(* PLC project Generated.project, CODESYS CODESYS V3.5 SP19 Patch 1 *)
(* stored: creationDateTime 2026-09-06T13:00:42.357406, modificationDateTime 2026-09-06T13:00:42.357406 *)

(* ======================================================================= 🔌 ST_ContactorCheck — Double vérification commande/retour contacteur ─────────────────────────────────────────────────────────────── 🎯 Rôle : Structure de diagnostic pour vérification commande vs retour 📊 Diagnostic : Détection des défauts contacteur (StuckClosed / StuckOpen) 📄 Doc métier : DOC/AF/AF_Partie-03_Contrats_Composants_v2.3.md §2 ======================================================================= *)
TYPE ST_ContactorCheck : STRUCT
  Command : BOOL;  (* Ordre envoyé au contacteur (TRUE = fermé/actif) *)
  Feedback : BOOL;  (* Retour d'état câblé (TRUE = effectivement fermé) *)
  StuckClosed : BOOL;  (* Diag : commande OFF mais retour ON depuis trop longtemps → PowerCutOff *)
  StuckOpen : BOOL;  (* Diag : commande ON mais retour OFF depuis trop longtemps *)
END_STRUCT;
END_TYPE

(* ======================================================================= 🧩 ST_Fault — Brique socle défaut (2 vues : live + latchée) ─────────────────────────────────────────────────────────────── 🎯 Rôle : porter l'état défaut d'un composant, applicable dans TOUS les cas (acquittable ou non), sans brique warning séparée. • Vue LIVE (Error / ErrorId) : suit la cause, retombe seule à 0. • Vue LATCHÉE (Latched / LatchedId): mémorisée au défaut, reste jusqu'au front Reset. Le choix acquittable / non-acquittable se fait PAR CAUSE (ST_FaultCause.Latching), jamais par bloc. 🔒 Sécurité : interlock TOUJOURS sur la cause brute (Error / ErrorId), jamais sur l'acquittement. Reset TOUJOURS effectif, jamais conditionné (std §9). 🧬 Composition : brique de base réutilisable — sortie de FB, struct métier, GVL. Texte IHM NON stocké ici : dérivé côté IHM depuis LatchedId / ErrorId. 📄 Doc : DOC/STDS/CODE_QUALITY_STANDARDS.md §2quinquies / §9 ======================================================================= *)
TYPE ST_Fault : STRUCT
  Error : BOOL;  (* <-- [DIAG] vue LIVE : au moins une cause présente maintenant *)
  ErrorId : WORD;  (* <-- [DIAG] bitfield des causes présentes maintenant (0 si aucune) *)
  Latched : BOOL;  (* <-- [DIAG] vue LATCHÉE : défaut non acquitté, reste jusqu'au front Reset *)
  LatchedId : WORD;  (* <-- [DIAG] ErrorId figé à l'apparition du défaut, effacé au Reset *)
END_STRUCT;
END_TYPE

(* ======================================================================= 🧩 ST_FaultCause — Cause élémentaire alimentant ST_Fault (socle FB_FaultCore) ─────────────────────────────────────────────────────────────── 🎯 Rôle : une cause exprimée EN CLAIR (BOOL + libellé), sans bitfield ni masque. Le FB métier remplit une liste (ARRAY[0..15] OF ST_FaultCause) ; le socle FB_FaultCore en déduit ST_Fault (vue live + vue latchée). 🔒 Sécurité : interlock TOUJOURS sur Active (cause brute), jamais sur le latch. Latching = TRUE → la cause ARME la vue latchée (défaut à acquitter). Latching = FALSE → la cause n'alimente que la vue live (retombe seule). Fail-safe : une cause laissée à Latching=FALSE reste visible en live — pour la rendre acquittable, il faut le déclarer explicitement. 📄 Doc : DOC/STDS/CODE_QUALITY_STANDARDS.md §2quinquies / §9 ======================================================================= *)
TYPE ST_FaultCause : STRUCT
  Active : BOOL;  (* 1 = cause présente maintenant (interlock sur cette valeur) *)
  Latching : BOOL;  (* 1 = cause à acquitter (arme Latched) ; 0 = live seulement *)
  Texte : STRING;  (* libellé prêt IHM (non stocké dans ST_Fault, dérivé côté IHM) *)
END_STRUCT;
END_TYPE

(* ======================================================================= 🛡️ FB_Brake — Séquence frein à manque de courant (temps physiques) ─────────────────────────────────────────────────────────────── 🎯 Rôle : Gestion temporisée ouverture/fermeture frein à manque de courant 🔒 Polarité : Sécurité positive (BrakeCmd=FALSE = frein collé au repos) 🔌 Interface : Double vérification retour contacteur (ST_ContactorCheck) 📄 Doc métier : DOC/AF/AF_Partie-10_Fonction_Winch_v2.1.md §3 ======================================================================= *)
FUNCTION_BLOCK FB_Brake
  VAR_INPUT
    Enable : BOOL;  (* === COMMANDES ET CONSIGNES === --> [CMD] Autorisation generale (FALSE = frein colle) *)
    Reset : BOOL;  (* --> [CMD] Acquittement defaut (front) *)
    MovementRequested : BOOL;  (* --> [CMD] Demande de mouvement (sens+palier actifs) *)
    ContactorFeedback : BOOL;  (* === RETOURS MATERIELS & SIMULATION === --> [HW] Retour contacteur frein (TRUE = relache/ouvert) *)
    BypassContactorCheck : BOOL;  (* --> [TST] Bypass controle contacteur (simu) *)
    DelayContactClose : TIME := TIME#100ms;  (* === TEMPORISATIONS ET REGLAGES === --> [CFG] Temps de fermeture contacteur de puissance *)
    DelayMagnetise : TIME := TIME#300ms;  (* --> [CFG] Delai magnetisation moteur avant ouverture frein *)
    DelayMotorDecel : TIME := TIME#500ms;  (* --> [CFG] Delai deceleration avant collage frein *)
    FeedbackTimeout : TIME := TIME#1s0ms;  (* --> [CFG] Delai max coherence commande/retour frein *)
  END_VAR
  VAR_OUTPUT
    Ready : BOOL;  (* === ETATS IEC & DERIVATION === <-- [STAT] FB pret a fonctionner *)
    Fault : ST_Fault;  (* 🧩 Statut transverse (forme cible ST_Fault) *)
    BrakeCmd : BOOL;  (* === COMMANDES ET CONFIRMATIONS === <-- [ACT] Commande bobine frein (TRUE = relache/ouvert) *)
    BrakeCommandOpenConfirmed : BOOL;  (* <-- [STAT] Confirmation ouverture frein pour verrous *)
    ContactorCheck : ST_ContactorCheck;  (* <-- [DIAG] Diagnostic detaille retour contacteur *)
  END_VAR
  VAR
    ResetEdge : R_TRIG;  (* === TRIGGERS ET DETECTION FRONTS === . [LOC] Detecteur front acquittement *)
    BypassEdge : R_TRIG;  (* . [LOC] Detecteur front activation bypass *)
    TonMagnetise : TON;  (* === TEMPORISATEURS INTERNES === . [LOC] Temporisation avant relachement frein *)
    TonDecel : TON;  (* . [LOC] Temporisation avant collage frein *)
    TonFeedback : TON;  (* . [LOC] Timeout de coherence commande/retour *)
    ContactorIncoherentError : BOOL;  (* === GESTION DES DEFAUTS === . [LOC] Défaut mémorisé incohérence contacteur *)
    instFault : FB_FaultCore;  (* * [INST] Socle de défaut *)
    instCauses : ARRAY[0..15] OF ST_FaultCause;  (* . [LOC] Table des causes nommées *)
  END_VAR

            

// === IMPLEMENTATION ===

{region "§1 Fronts"}
// 🔑 1. FRONTS
ResetEdge(CLK := Reset);
BypassEdge(CLK := BypassContactorCheck);

// Acquittement des drapeaux contacteur
IF ResetEdge.Q OR BypassContactorCheck THEN
    ContactorIncoherentError := FALSE;
    ContactorCheck.StuckClosed := FALSE;
    ContactorCheck.StuckOpen   := FALSE;
END_IF;
{endregion}

{region "§2 Gate neutralisation"}
// 🛑 2. GATE — pas d'Enable = frein collé (sécurité positive), aucune temporisation en cours
IF NOT Enable THEN
    TonMagnetise(IN := FALSE, PT := DelayMagnetise + DelayContactClose);
    TonDecel(IN := FALSE, PT := DelayMotorDecel);
    TonFeedback(IN := FALSE, PT := FeedbackTimeout);
    BrakeCmd := FALSE;
    Ready := FALSE;
    ContactorCheck.Command := FALSE;          // 📊 Neutralisation : miroir de BrakeCmd := FALSE
    ContactorCheck.Feedback := ContactorFeedback; // 📊 Neutralisation : miroir entrée physique
    BrakeCommandOpenConfirmed := FALSE;       // 🛡️ Fail-Safe : frein commandé fermé hors Enable
    
    // Évaluation du socle de défaut sous neutralisation (permet acquittement Reset hors Enable)
    instCauses[0].Active   := FALSE;
    instCauses[0].Latching := TRUE;
    instCauses[0].Texte    := 'Incoherence retour contacteur frein';
    instFault(Enable := FALSE, Reset := Reset, Causes := instCauses);
    Fault := instFault.Fault;
    RETURN;
END_IF;
{endregion}

{region "§3 Séquence temporisée"}
// 🛠️ 3. SÉQUENCE TEMPORISÉE (démarrage vs arrêt)
IF MovementRequested THEN
    TonDecel(IN := FALSE, PT := DelayMotorDecel);
    TonMagnetise(IN := TRUE, PT := DelayMagnetise + DelayContactClose);
    IF TonMagnetise.Q THEN
        BrakeCmd := TRUE;              // ✅ Contacteur + magnétisation acquis → relâche
    ELSE
        BrakeCmd := FALSE;             // ⏳ Encore collé pendant la magnétisation
    END_IF;
ELSE
    // Sécurité positive : fermeture immédiate du frein (collé) dès que les contacteurs de sens s'ouvrent
    TonMagnetise(IN := FALSE, PT := DelayMagnetise + DelayContactClose);
    TonDecel(IN := FALSE, PT := DelayMotorDecel);
    BrakeCmd := FALSE;                 // Fermeture immédiate
END_IF;
{endregion}

{region "§4 Double vérification contacteur"}
// 🔍 4. DOUBLE VÉRIFICATION RETOUR CONTACTEUR (ST_ContactorCheck)
ContactorCheck.Command := BrakeCmd;
ContactorCheck.Feedback := ContactorFeedback;

// ContactorFeedback est dans le MÊME sens que BrakeCmd (TRUE = relâché = frein ouvert).
TonFeedback(IN := (BrakeCmd <> ContactorFeedback), PT := FeedbackTimeout);
IF NOT BypassContactorCheck THEN
    IF TonFeedback.Q THEN
        ContactorCheck.StuckClosed := (BrakeCmd AND NOT ContactorFeedback);
        ContactorCheck.StuckOpen   := (NOT BrakeCmd AND ContactorFeedback);
        ContactorIncoherentError   := TRUE;
    END_IF;
END_IF;
{endregion}

{region "§5 Causes & Socle Défaut"}
// 🚨 5. SOCLE DÉFAUT & SORTIE SÛRE
instCauses[0].Active   := NOT BypassContactorCheck AND (ContactorCheck.StuckClosed OR ContactorCheck.StuckOpen OR (TonFeedback.Q AND (BrakeCmd <> ContactorFeedback)));
instCauses[0].Latching := TRUE;
instCauses[0].Texte    := 'Incoherence retour contacteur frein';

instFault(Enable := Enable, Reset := Reset, Causes := instCauses);
Fault := instFault.Fault;

Ready := Enable AND NOT Fault.Latched;

// Sortie sûre immédiate
IF Fault.Error OR Fault.Latched THEN
    BrakeCmd := FALSE;
END_IF;
{endregion}

{region "§6 Confirmation ouverture"}
// 📤 6. CONFIRMATION OUVERTURE FREIN
IF BypassContactorCheck THEN
    BrakeCommandOpenConfirmed := BrakeCmd;
ELSE
    BrakeCommandOpenConfirmed := ContactorFeedback AND NOT Fault.Latched;  (* TRUE = frein ouvert = desserrage confirmé *)
END_IF;
{endregion}

          
END_FUNCTION_BLOCK

(* ======================================================================= 🧩 FB_FaultCore — Socle de remplissage de ST_Fault (vue live + vue latchée) ─────────────────────────────────────────────────────────────── 🎯 Rôle : à partir d'une LISTE de causes en clair (ARRAY[0..15] OF ST_FaultCause), produire la brique ST_Fault : • Error / ErrorId : vue LIVE, suit les causes Active, retombe seule. • Latched / LatchedId: vue LATCHÉE, chaque bit figé à l'apparition d'une cause `Active AND Latching`, conservé jusqu'au front Reset. 🔒 Sécurité : - interlock TOUJOURS sur `Causes[i].Active` (cause brute), jamais sur le latch. - Reset TOUJOURS effectif, jamais conditionné (std §9) — agit même Enable=FALSE. - Latching=FALSE → cause visible en LIVE seulement (fail-safe : reste visible). - un défaut laté non acquitté reste publié même FB désactivé (pas d'effacement silencieux sur bascule Enable OFF→ON sans Reset). - une cause à acquitter réapparue re-arme son bit (ré-alarme). 🧬 Un seul socle, réutilisé par tout FB `standard` qui expose un ST_Fault. Pas de State, pas de Warning, pas de texte — hors périmètre de ce socle. 📄 Doc : DOC/STDS/CODE_QUALITY_STANDARDS.md §2quinquies / §9 ======================================================================= *)
FUNCTION_BLOCK FB_FaultCore
  VAR_INPUT
    Enable : BOOL;  (* --> [CMD] Autorisation générale du FB porteur *)
    Reset : BOOL;  (* --> [CMD] Front d'acquittement (jamais conditionné, §9) *)
    Causes : ARRAY[0..15] OF ST_FaultCause;  (* --> [CMD] Liste des causes en clair (Active / Latching / Texte) *)
  END_VAR
  VAR_OUTPUT
    Ready : BOOL;  (* <-- [STAT] FB porteur autorisé (= Enable) *)
    Fault : ST_Fault;  (* <-- [DIAG] Brique défaut (mappée 1:1 sur la sortie du FB porteur) *)
  END_VAR
  VAR
    ResetEdge : R_TRIG;  (* . [LOC] Front montant Reset *)
    Latch : ARRAY[0..15] OF BOOL;  (* . [LOC] Bit laté par cause, jusqu'au Reset *)
    i : INT;  (* . [LOC] Index de parcours de la liste *)
  END_VAR

            

{region "§1 Reset (front, toujours effectif)"}
// Front Reset : efface tous les latches. Jamais conditionné, agit même Enable=FALSE (§9).
Ready := Enable;
ResetEdge(CLK := Reset);
IF ResetEdge.Q THEN
    FOR i := 0 TO 15 DO Latch[i] := FALSE; END_FOR;
END_IF;
{endregion}

{region "§2 Vue LIVE — Error / ErrorId"}
// Bitfield des causes présentes MAINTENANT. Retombe seule à 0 quand les causes disparaissent.
// Non évaluée si Enable=FALSE (pas de lecture de cause hors autorisation).
Fault.ErrorId := 0;
IF Enable THEN
    FOR i := 0 TO 15 DO
        IF Causes[i].Active THEN
            Fault.ErrorId := Fault.ErrorId OR SHL(WORD#1, INT_TO_DWORD(i));
        END_IF;
    END_FOR;
END_IF;
Fault.Error := (Fault.ErrorId <> 0);
{endregion}

{region "§3 Armement des latches (causes à acquitter)"}
// Une cause Active ET Latching arme son bit ; le bit reste jusqu'au front Reset (§1),
// même si la cause disparaît. Réapparition => ré-armement (ré-alarme).
IF Enable THEN
    FOR i := 0 TO 15 DO
        IF Causes[i].Active AND Causes[i].Latching THEN
            Latch[i] := TRUE;
        END_IF;
    END_FOR;
END_IF;
{endregion}

{region "§4 Vue LATCHÉE — Latched / LatchedId"}
// Toujours publiée, y compris Enable=FALSE : un défaut non acquitté reste visible.
Fault.LatchedId := 0;
FOR i := 0 TO 15 DO
    IF Latch[i] THEN
        Fault.LatchedId := Fault.LatchedId OR SHL(WORD#1, INT_TO_DWORD(i));
    END_IF;
END_FOR;
Fault.Latched := (Fault.LatchedId <> 0);
{endregion}

          
END_FUNCTION_BLOCK
